FUNCTION HLI3_FindHliAxisIdx : DINT
VAR_INPUT
	nLogAxisNo		: UDINT;	
END_VAR
VAR
	i				: UINT;	
END_VAR

IF nLogAxisNo > MAX_SYS_LOG_AXIS_INDEX OR nLogAxisNo < 1 THEN 
	HLI3_FindHliAxisIdx := -1;
ELSE
	HLI3_FindHliAxisIdx := CNCSystem.LogAxisNo[nLogAxisNo].nHliAxisIdx;	
END_IF

END_FUNCTION

(* stored: Version 1.1.0.1, ProductVersion 3.1.4018.5
   POU HLI3_FindHliAxisIdx: Id {7aa33349-5577-41f0-8d51-fe242c595c7e}, SpecialFunc None *)
